(* Schneider Machine Expert - Basic project UNO_pipe_new_ip (1), file version 2.0.0.0 *)
(* ProjectInformations: Name=New project *)
(* UserInformations: LastName=GORDON, FirstName=JOHN, PhoneNumber=205-679-4000 *)

HARDWARE
  Cpu 0: TM221CE16R
  ModuleExtensionObject 0: TM3AM6/G
  EthernetConfiguration: NetworkName=M221, IpAllocationMode=FixedAddress, IpAddress=10.10.0.131, SubnetMask=255.255.0.0
  SerialLineConfiguration: Baud=Baud19200, Parity=ParityEven, DataBits=DataBits8, StopBits=StopBits1, PhysicalMedium=PhysicalMediumRs485, TransmissionMode=TransmissionModeModbusRtu, SlaveId=1, Addressing=SlaveAddressing
  MastTask: UsePeriodScanMode=false, PeriodScan=100
  FastTask: Period=255
  CpuBehavior: StartingMode=StartInRun, AutoSaveRamOnEeprom=true, WatchdogPeriod=250

SYMBOLS  (address, symbol, comment, settings)
  %M0       SYSTEM_RUN  "0=OFF, 1=ON"
  %M1       SOLENOID_ON  "Solenoid Open Command"
  %M2       PUMP_ON  "Air Pump Run Command"
  %M4       POWER_ON
  %M5       FORCE_ON  "1"
  %M7       FORCED_ON_AIR
  %M10      FIRST_SCAN
  %MW0      HMI_PRESS_SP_HI  "High Pressure Setpoint set from HMI"
  %MW1      HMI_PRESS_SP_LO  "Low Pressure Setpoint set from HMI"
  %MF0      PRESSURE
  %TM0      AIR_BLEED_TIMER  "Air Bleed Timer"  [Type=TP, Preset=5, Base=OneSecond]
  %I0.0     PRESSURE_SW_INPUT
  %Q0.0     AIR_PUMP_RUN
  %Q0.1     SOLENOID_OPEN
  %QWE0     PRESSURE_SIGNAL_EIP
  %IW1.0    PRESSURE_SIGNAL  [Type=Type_4_20mA, Scope=Scope_Customized, Minimum=0, Maximum=1450]

POU New POU
  (* SectionNumber=1 *)

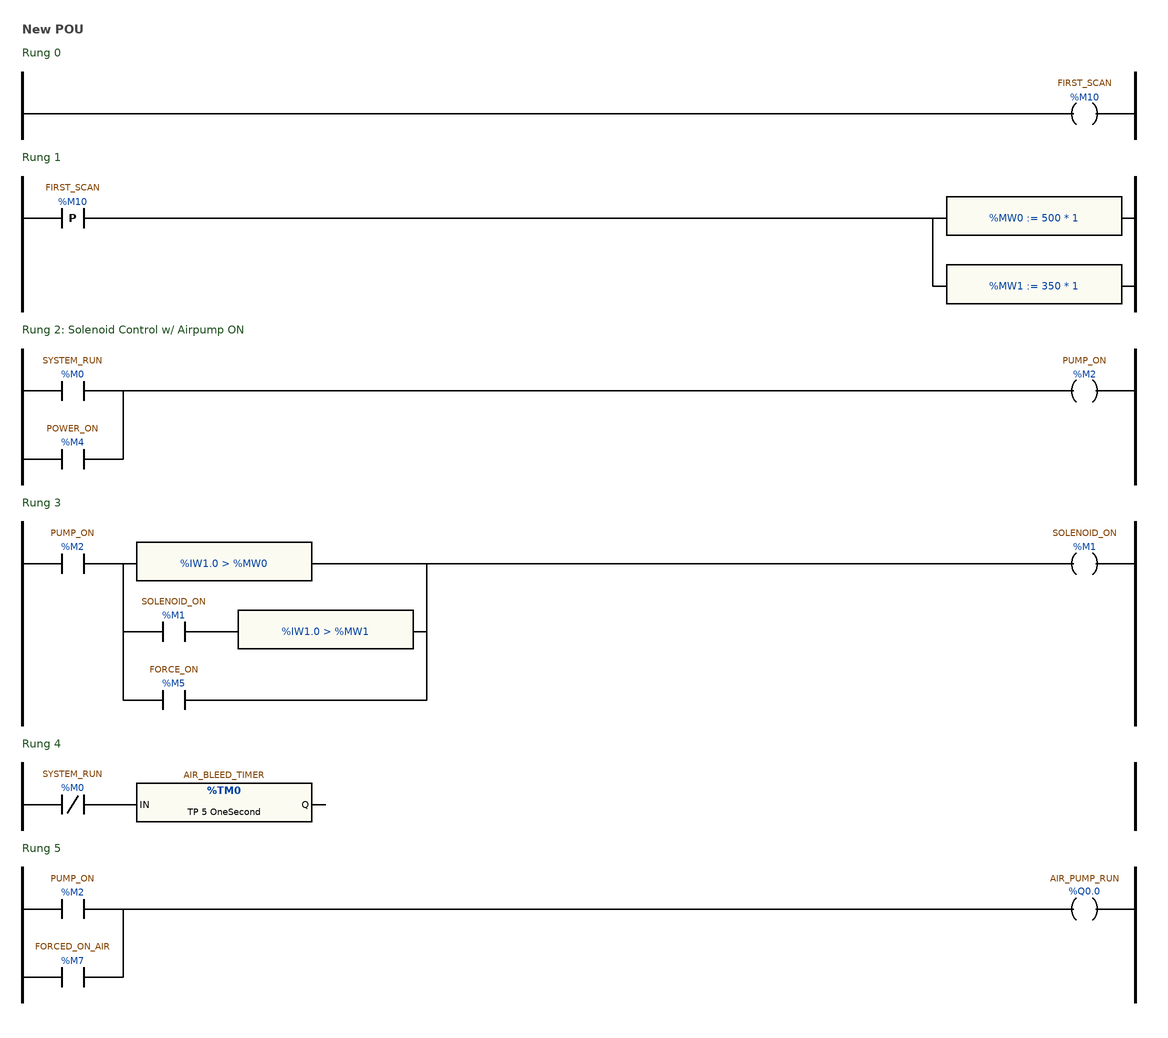

// Rung 0
  LD 1
  ST %M10                 (* FIRST_SCAN *)
  // as ST:
  //   FIRST_SCAN := TRUE;

// Rung 1
  LDR %M10                (* FIRST_SCAN *)
  [ %MW0 := 500 * 1 ]     (* HMI_PRESS_SP_HI *)
  [ %MW1 := 350 * 1 ]     (* HMI_PRESS_SP_LO *)
  // as ST:
  //   IF RISING(FIRST_SCAN) THEN HMI_PRESS_SP_HI := 500 * 1; END_IF;
  //   IF RISING(FIRST_SCAN) THEN HMI_PRESS_SP_LO := 350 * 1; END_IF;

// Rung 2: Solenoid Control w/ Airpump ON
  LD %M0                  (* SYSTEM_RUN *)
  OR %M4                  (* POWER_ON *)
  ST %M2                  (* PUMP_ON *)
  // as ST:
  //   PUMP_ON := SYSTEM_RUN OR POWER_ON;

// Rung 3
  LD %M2                  (* PUMP_ON *)
  AND( [ %IW1.0 > %MW0 ]  (* PRESSURE_SIGNAL, HMI_PRESS_SP_HI *)
  OR( %M1                 (* SOLENOID_ON *)
  AND [ %IW1.0 > %MW1 ]   (* PRESSURE_SIGNAL, HMI_PRESS_SP_LO *)
  )
  OR %M5                  (* FORCE_ON *)
  )
  ST %M1                  (* SOLENOID_ON *)
  // as ST:
  //   SOLENOID_ON := PUMP_ON AND (PRESSURE_SIGNAL > HMI_PRESS_SP_HI OR SOLENOID_ON AND PRESSURE_SIGNAL > HMI_PRESS_SP_LO OR FORCE_ON);

// Rung 4
  BLK %TM0                (* AIR_BLEED_TIMER *)
  LDN %M0                 (* SYSTEM_RUN *)
  IN
  END_BLK
  // as ST:
  //   AIR_BLEED_TIMER(IN := NOT SYSTEM_RUN);

// Rung 5
  LD %M2                  (* PUMP_ON *)
  OR %M7                  (* FORCED_ON_AIR *)
  ST %Q0.0                (* AIR_PUMP_RUN *)
  // as ST:
  //   AIR_PUMP_RUN := PUMP_ON OR FORCED_ON_AIR;

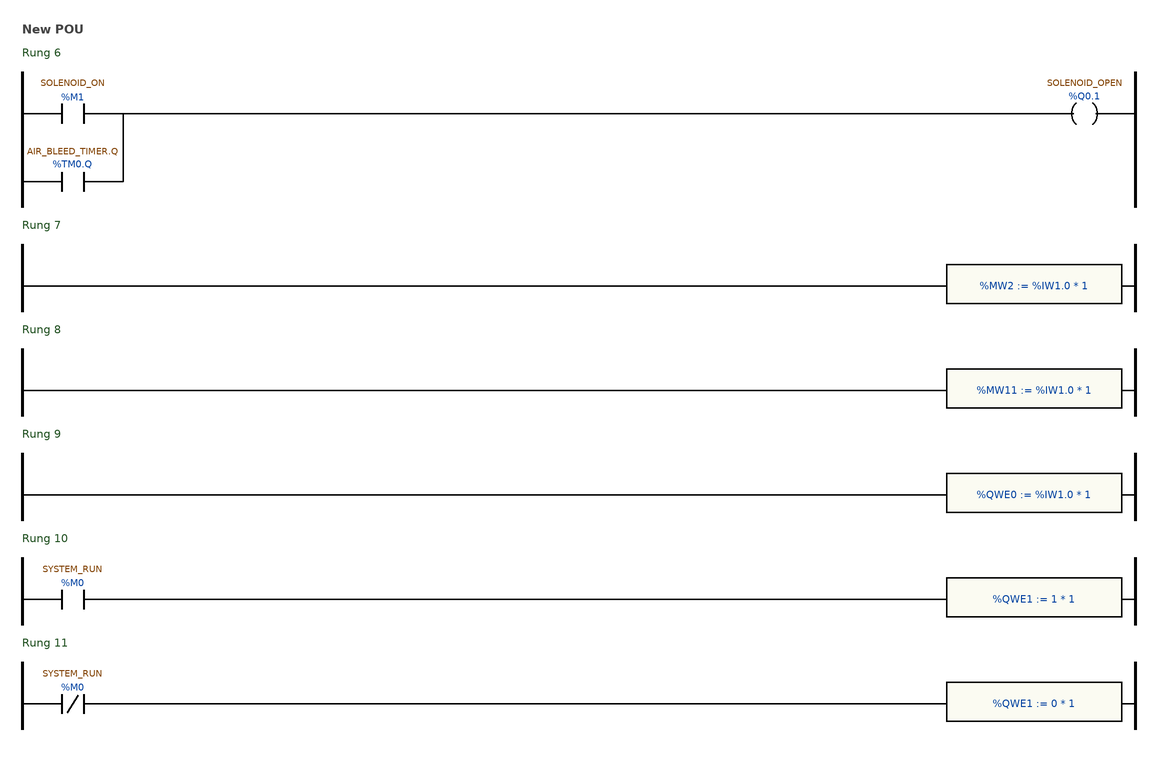

// Rung 6
  LD %M1                  (* SOLENOID_ON *)
  OR %TM0.Q               (* AIR_BLEED_TIMER *)
  ST %Q0.1                (* SOLENOID_OPEN *)
  // as ST:
  //   SOLENOID_OPEN := SOLENOID_ON OR AIR_BLEED_TIMER.Q;

// Rung 7
  LD 1
  [ %MW2 := %IW1.0 * 1 ]  (* PRESSURE_SIGNAL *)
  // as ST:
  //   %MW2 := PRESSURE_SIGNAL * 1;

// Rung 8
  LD 1
  [ %MW11 := %IW1.0 * 1 ] (* PRESSURE_SIGNAL *)
  // as ST:
  //   %MW11 := PRESSURE_SIGNAL * 1;

// Rung 9
  LD 1
  [ %QWE0 := %IW1.0 * 1 ] (* PRESSURE_SIGNAL_EIP, PRESSURE_SIGNAL *)
  // as ST:
  //   PRESSURE_SIGNAL_EIP := PRESSURE_SIGNAL * 1;

// Rung 10
  LD %M0                  (* SYSTEM_RUN *)
  [ %QWE1 := 1 * 1 ]
  // as ST:
  //   IF SYSTEM_RUN THEN %QWE1 := 1 * 1; END_IF;

// Rung 11
  LDN %M0                 (* SYSTEM_RUN *)
  [ %QWE1 := 0 * 1 ]
  // as ST:
  //   IF NOT SYSTEM_RUN THEN %QWE1 := 0 * 1; END_IF;
